FUNCTION_BLOCK T_RoboConnect_SetAnalogOutput_IncorrectIndexFails EXTENDS T_UnitTestBase
VAR
  robot : I_RoboConnect;
  targetDO : UINT;
  myTestState, prevState :
    (INIT, ARRANGE, ACT, ASSERT) := INIT;
  expected: BOOL;
  actual : BOOL := TRUE;
  counter : UINT;
END_VAR

CASE myTestState OF
  INIT:
    StateChanged();
    myTestState := ARRANGE;

  ARRANGE:
    IF StateChanged() THEN
      expected := FALSE;
      myTestState := ACT;
    END_IF

  ACT:
    actual := robot.SetAnalogOutput(targetDO, 0.5);
    myTestState := ASSERT;

  ASSERT:
    assertion.AssertEquals_BOOL(expected, actual, 'robot.SetAnalogOutput(targetDO,TRUE)');
    TestFinished();
    myTestState := INIT;

END_CASE

METHOD FB_init : BOOL
VAR_INPUT
  bInitRetains : BOOL; // if TRUE, the retain variables are initialized (warm start / cold start)
  bInCopyCode : BOOL; // if TRUE, the instance afterwards gets moved into the copy code (online change)
  TestSuite : tcl_SimpleUnitTestLibrary.I_TestSuite;
  robot : I_TcRobot;
  targetDo : UINT;
END_VAR
THIS^.robot := robot;
THIS^.targetDo := targetDo;
END_METHOD

METHOD PRIVATE StateChanged : BOOL
IF  myTestState = prevState THEN
  RETURN;
END_IF

prevState := myTestState;
StateChanged := TRUE;
END_METHOD

METHOD WaitForCycles : BOOL
VAR_INPUT
  maxCount : UINT;
END_VAR
counter := counter + 1;

IF counter = maxCount THEN
  counter := 0;
  WaitForCycles := TRUE;
END_IF
END_METHOD

END_FUNCTION_BLOCK

(* stored: Version 1.1.0.1
   POU T_TcRobot_SetAnalogOutput_IncorrectIndexFails: Id {e2c7152e-3137-4385-a83c-540e4744b3fa}, SpecialFunc None
   Method FB_init: Id {a2f15066-30cc-4036-ba6c-0588bc1818ec}
   Method StateChanged: Id {16d7f861-c8b9-4e41-9af2-2a648325b71c}
   Method WaitForCycles: Id {eacc52c5-2185-4a59-8337-6be53c7e0fa4} *)
